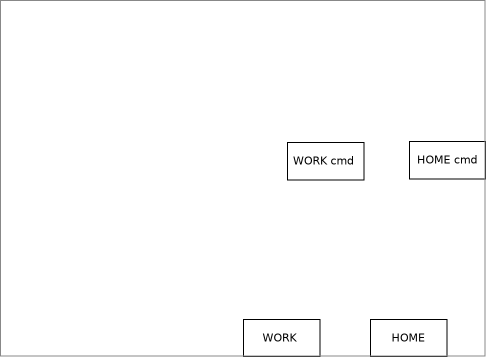
VISUALIZATION Visualization  // 486x357
    Rectangle (287,142 77x38), "WORK cmd"
    Rectangle (409,141 77x38), "HOME cmd"
    Rectangle (243,319 77x38), "WORK"
    Rectangle (370,319 77x38), "HOME"
END_VISUALIZATION

(* stored: Version 1.1.0.1, ProductVersion 3.1.4024.16
   Visu Visualization: Id {8a892678-d7da-4d9a-ba18-8b474e0be024} *)
